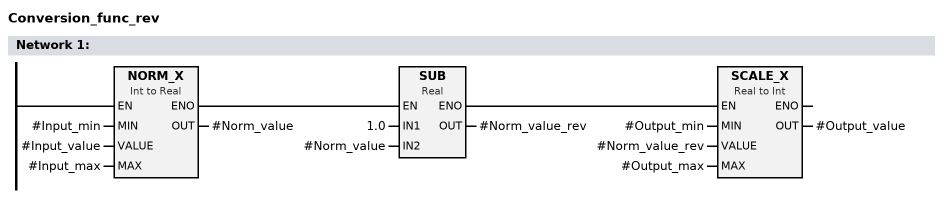
   RUNG wire#powerrail
      { S7_Templates := "[SrcType := Int, DestType := Real]" } Normalize(min := #Input_min, value := #Input_value, max := #Input_max, out => #Norm_value)
      { S7_Templates := "SrcType := Real" } Sub(in1 := 1.0, in2 := #Norm_value, out => #Norm_value_rev)
      { S7_Templates := "[SrcType := Real, DestType := Int]" } Scale(min := #Output_min, value := #Norm_value_rev, max := #Output_max, out => #Output_value)
   END_RUNG
   // the same network as SCL:
   #Norm_value := NORM_X(MIN := #Input_min, VALUE := #Input_value, MAX := #Input_max);
   #Norm_value_rev := 1.0 - #Norm_value;
   #Output_value := SCALE_X(MIN := #Output_min, VALUE := #Norm_value_rev, MAX := #Output_max);
END_REGION
END_FUNCTION

ORGANIZATION_BLOCK "Main"   // OB1, LAD, ProgramCycle
TITLE = "Main Program Sweep (Cycle)"
{ S7_Optimized_Access := 'TRUE' }
VERSION : 0.1
// Main program here to manage and call all FBs and FCs.
   VAR_INPUT
      Initial_Call : Bool;   // Initial call of this OB
      Remanence : Bool;   // =True, if remanent data are available
   END_VAR
   VAR_TEMP
      SequenceInit : Bool;
      InitSequence : Bool;
      Language : Int;
   END_VAR
   VAR_TEMP   // added for the SCL form of the ladder/FBD networks
      _w1 : Bool;
      _w2 : Bool;
      _w3 : Bool;
      _w4 : Bool;
   END_VAR
BEGIN

REGION Network 1: Call the simulation block.
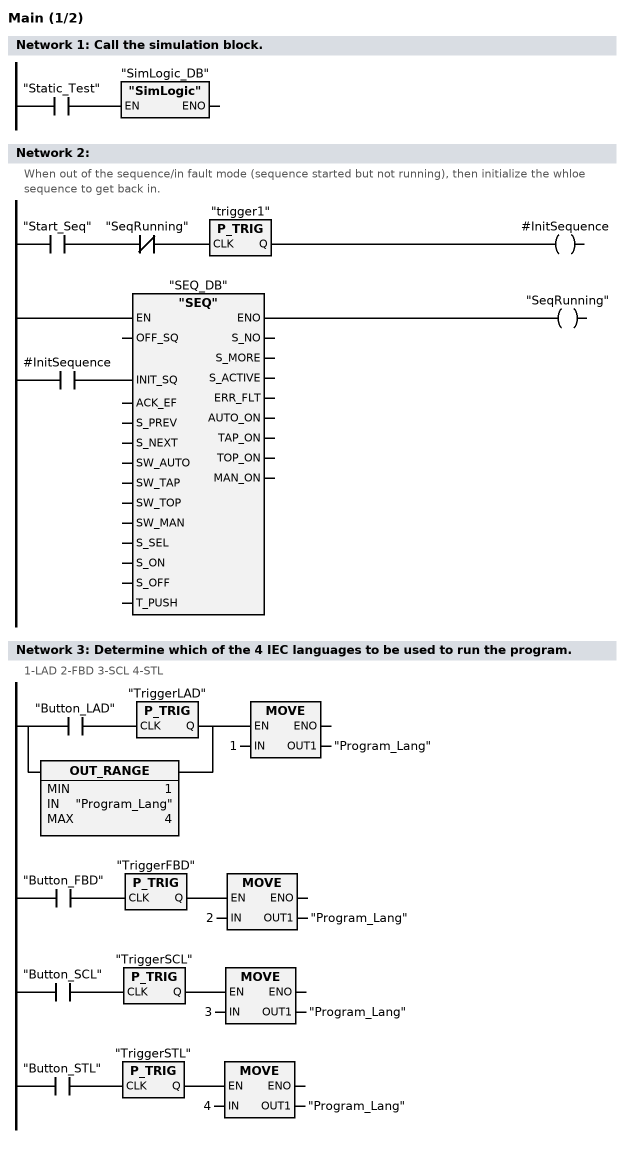
   RUNG wire#powerrail
      Contact( "Static_Test" )
      "SimLogic_DB"()
   END_RUNG
   // the same network as SCL:
   IF "Static_Test" THEN
       "SimLogic_DB"();   // "SimLogic"
   END_IF;
END_REGION

REGION Network 2
   // When out of the sequence/in fault mode (sequence started but not running), then initialize the whloe sequence to get back in.
   RUNG wire#powerrail
      Contact( "Start_Seq" )
      I_Contact( "SeqRunning" )
      P_Trig( "trigger1" )
      Coil( #InitSequence )
   END_RUNG
   RUNG wire#powerrail
      "SEQ_DB"(INIT_SQ := wire#w1, OFF_SQ :=, ACK_EF :=, S_PREV :=, S_NEXT :=, SW_AUTO :=, SW_TAP :=, SW_TOP :=, SW_MAN :=, S_SEL :=, S_ON :=, S_OFF :=, T_PUSH :=, S_NO =>, S_MORE =>, S_ACTIVE =>, ERR_FLT =>, AUTO_ON =>, TAP_ON =>, TOP_ON =>, MAN_ON =>)
      Coil( "SeqRunning" )
   END_RUNG
   RUNG wire#powerrail
      Contact( #InitSequence )
   END_RUNG wire#w1
   // the same network as SCL:
   #_w1 := "Start_Seq" AND NOT "SeqRunning";
   #_w2 := #_w1 AND NOT "trigger1";   // rising edge
   "trigger1" := #_w1;
   #InitSequence := #_w2;
   "SEQ_DB"(INIT_SQ := #InitSequence, ENO => #_w3);   // "SEQ"
   "SeqRunning" := #_w3;
END_REGION

REGION Network 3: Determine which of the 4 IEC languages to be used to run the program.
   // 1-LAD 2-FBD 3-SCL 4-STL
   #_w1 := "Button_LAD" AND NOT "TriggerLAD";   // rising edge
   "TriggerLAD" := "Button_LAD";
   IF #_w1 OR ("Program_Lang" < 1) OR ("Program_Lang" > 4) THEN "Program_Lang" := 1; END_IF;
   #_w2 := "Button_FBD" AND NOT "TriggerFBD";   // rising edge
   "TriggerFBD" := "Button_FBD";
   IF #_w2 THEN "Program_Lang" := 2; END_IF;
   #_w3 := "Button_SCL" AND NOT "TriggerSCL";   // rising edge
   "TriggerSCL" := "Button_SCL";
   IF #_w3 THEN "Program_Lang" := 3; END_IF;
   #_w4 := "Button_STL" AND NOT "TriggerSTL";   // rising edge
   "TriggerSTL" := "Button_STL";
   IF #_w4 THEN "Program_Lang" := 4; END_IF;
END_REGION

REGION Network 4: When a language is chosen, run the corresponding program.
   // 1-LAD 2-FBD 3-SCL 4-STL
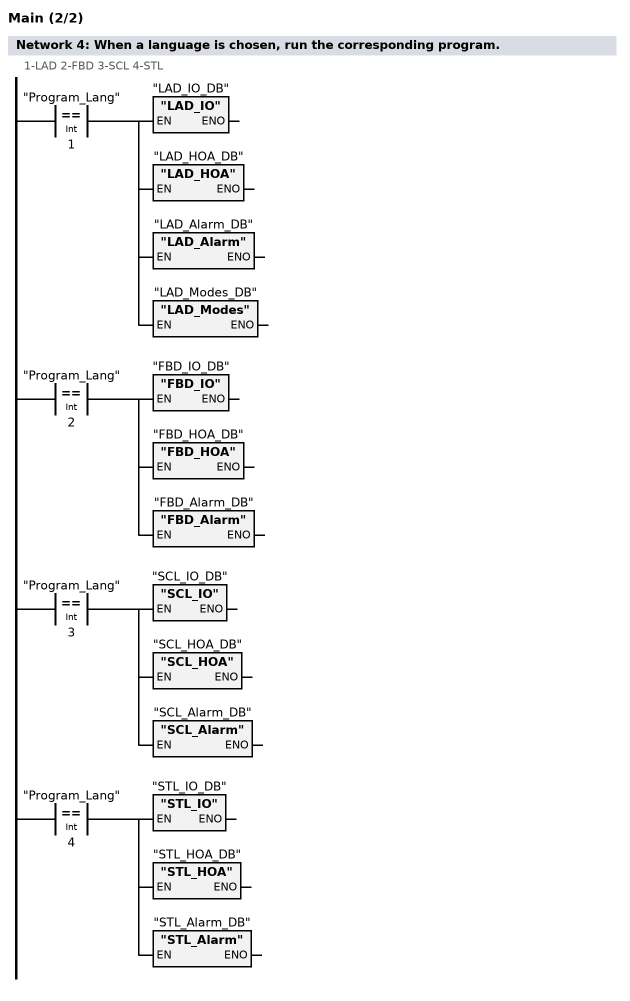
   RUNG wire#powerrail
      { S7_Templates := "SrcType := Int" } EQ_Contact(in1 := "Program_Lang", in2 := 1)
      wire#w1
      "LAD_IO_DB"()
   END_RUNG
   RUNG wire#w1
      "LAD_HOA_DB"()
   END_RUNG
   RUNG wire#w1
      "LAD_Alarm_DB"()
   END_RUNG
   RUNG wire#w1
      "LAD_Modes_DB"()
   END_RUNG
   RUNG wire#powerrail
      { S7_Templates := "SrcType := Int" } EQ_Contact(in1 := "Program_Lang", in2 := 2)
      wire#w2
      "FBD_IO_DB"()
   END_RUNG
   RUNG wire#w2
      "FBD_HOA_DB"()
   END_RUNG
   RUNG wire#w2
      "FBD_Alarm_DB"()
   END_RUNG
   RUNG wire#powerrail
      { S7_Templates := "SrcType := Int" } EQ_Contact(in1 := "Program_Lang", in2 := 3)
      wire#w3
      "SCL_IO_DB"()
   END_RUNG
   RUNG wire#w3
      "SCL_HOA_DB"()
   END_RUNG
   RUNG wire#w3
      "SCL_Alarm_DB"()
   END_RUNG
   RUNG wire#powerrail
      { S7_Templates := "SrcType := Int" } EQ_Contact(in1 := "Program_Lang", in2 := 4)
      wire#w4
      "STL_IO_DB"()
   END_RUNG
   RUNG wire#w4
      "STL_HOA_DB"()
   END_RUNG
   RUNG wire#w4
      "STL_Alarm_DB"()
   END_RUNG
   // the same network as SCL:
   #_w1 := "Program_Lang" = 1;
   IF #_w1 THEN
       "LAD_IO_DB"();   // "LAD_IO"
       "LAD_HOA_DB"();   // "LAD_HOA"
       "LAD_Alarm_DB"();   // "LAD_Alarm"
       "LAD_Modes_DB"();   // "LAD_Modes"
   END_IF;
   #_w2 := "Program_Lang" = 2;
   IF #_w2 THEN
       "FBD_IO_DB"();   // "FBD_IO"
       "FBD_HOA_DB"();   // "FBD_HOA"
       "FBD_Alarm_DB"();   // "FBD_Alarm"
   END_IF;
   #_w3 := "Program_Lang" = 3;
   IF #_w3 THEN
       "SCL_IO_DB"();   // "SCL_IO"
       "SCL_HOA_DB"();   // "SCL_HOA"
       "SCL_Alarm_DB"();   // "SCL_Alarm"
   END_IF;
   #_w4 := "Program_Lang" = 4;
   IF #_w4 THEN
       "STL_IO_DB"();   // "STL_IO"
       "STL_HOA_DB"();   // "STL_HOA"
       "STL_Alarm_DB"();   // "STL_Alarm"
   END_IF;
END_REGION
END_ORGANIZATION_BLOCK

ORGANIZATION_BLOCK "PID"   // OB30, LAD, CyclicInterrupt
{ S7_Optimized_Access := 'TRUE' }
VERSION : 0.1
   VAR_INPUT
      Initial_Call : Bool;   // Initial call of this OB
      Event_Count : Int;   // Events discarded
   END_VAR
   VAR_TEMP   // added for the SCL form of the ladder/FBD networks
      _w1 : Bool;
   END_VAR
BEGIN

REGION Network 1
   // High oil flow alarm handling
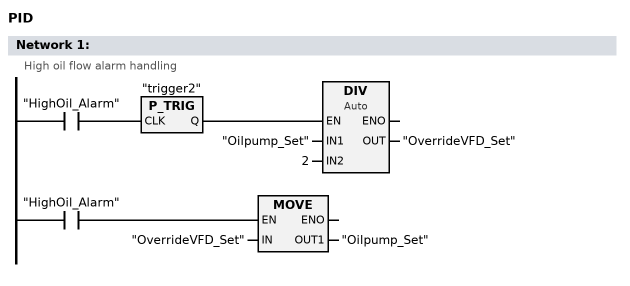
   RUNG wire#powerrail
      Contact( "HighOil_Alarm" )
      P_Trig( "trigger2" )
      Div(in1 := "Oilpump_Set", in2 := 2, out => "OverrideVFD_Set")
   END_RUNG
   RUNG wire#powerrail
      Contact( "HighOil_Alarm" )
      Move(in := "OverrideVFD_Set", out1 => "Oilpump_Set")
   END_RUNG
   // the same network as SCL:
   #_w1 := "HighOil_Alarm" AND NOT "trigger2";   // rising edge
   "trigger2" := "HighOil_Alarm";
   IF #_w1 THEN "OverrideVFD_Set" := "Oilpump_Set" / 2; END_IF;
   IF "HighOil_Alarm" THEN "Oilpump_Set" := "OverrideVFD_Set"; END_IF;
END_REGION
END_ORGANIZATION_BLOCK

(* ===== HMI "HMI_RT_1" =====
connection "HMI_Connection_1": ETHERNET, S7_1500_OMS
*)